# EPICS substitutions: ek9000App/Db/EL1814_mbbiDirect.substitutions
file EL1814.template
{       pattern
        {
                TERMINAL,

        }
        {
        }
}
